FUNCTION_BLOCK STATION3_INFO
  {SET_ATTRIBUTE(OpcUa, SERVICE)}
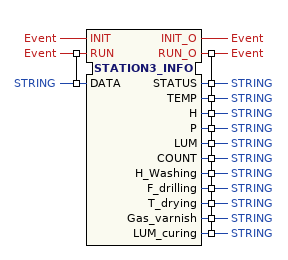
  EVENT_INPUT
    INIT;
    RUN WITH DATA; {SET_ATTRIBUTE(OpcUa, Method)}
  END_EVENT
  EVENT_OUTPUT
    INIT_O;
    RUN_O WITH STATUS, TEMP, H, P, LUM, COUNT, H_Washing, F_drilling, T_drying, Gas_varnish, LUM_curing;
  END_EVENT
  VAR_INPUT
    DATA : STRING;
  END_VAR
  VAR_OUTPUT
    STATUS : STRING;
    TEMP : STRING;
    H : STRING;
    P : STRING;
    LUM : STRING;
    COUNT : STRING;
    H_Washing : STRING;
    F_drilling : STRING;
    T_drying : STRING;
    Gas_varnish : STRING;
    LUM_curing : STRING;
  END_VAR
END_FUNCTION_BLOCK
